// TIA Portal V17 export
// export: Created 2021-12-03T08:13:11.653875Z, ExportSetting WithDefaults, DisplayName Totally Integrated Automation Portal, DisplayVersion V17, DisplayName TIA Portal Openness, DisplayVersion V17, DisplayName TIA Portal Version Control Interface, DisplayVersion V17, DisplayName STEP 7 Professional, DisplayVersion V17, DisplayName STEP 7 Safety, DisplayVersion V17, DisplayName WinCC Advanced, DisplayVersion V17
FUNCTION "FFC_ContCtrl" : Void   // FC700, F_FBD
VERSION : 0.1
// stored: AutoNumber false, IsIECCheckEnabled false, UDAEnableTagReadback false
BEGIN

REGION Network 2: Таймер на включение 400В через 15 секунд после 230В / Задержка между включением 230 и 380 В
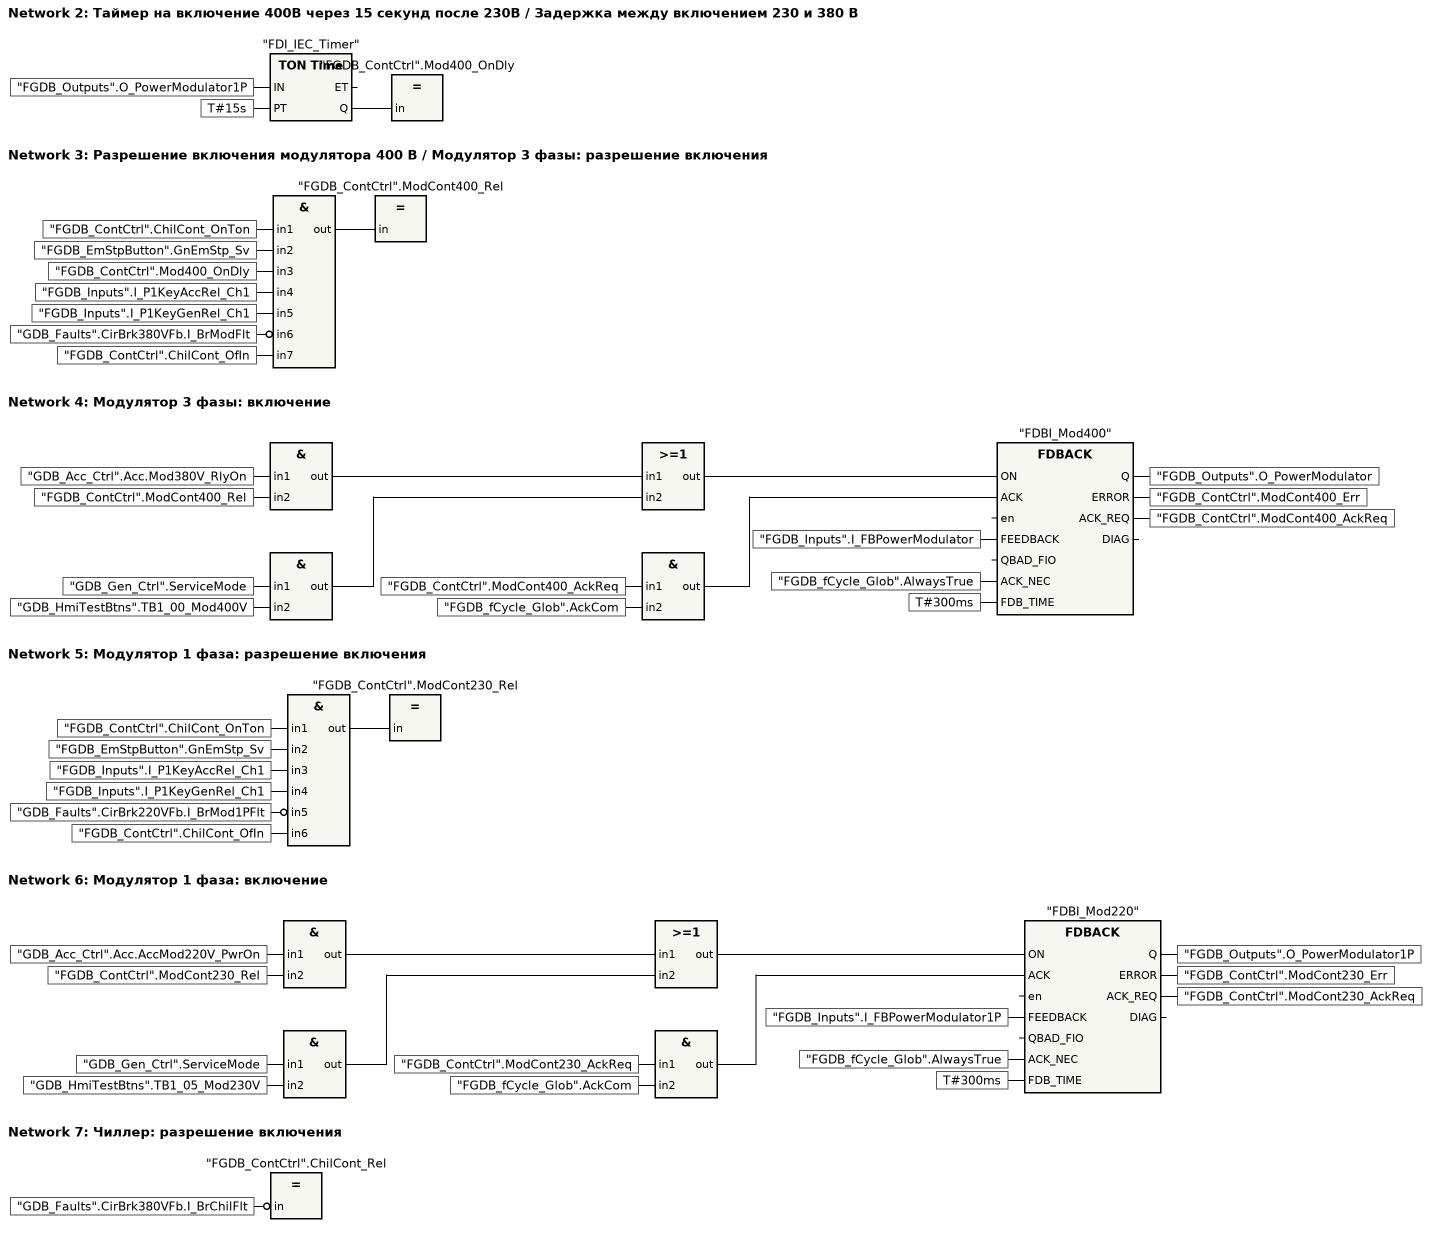
   "FDI_IEC_Timer".TON(IN := "FGDB_Outputs".O_PowerModulator1P, PT := T#15s);
   "FGDB_ContCtrl".Mod400_OnDly := "FDI_IEC_Timer".Q;
END_REGION

REGION Network 3: Разрешение включения модулятора 400 В / Модулятор 3 фазы: разрешение включения
   "FGDB_ContCtrl".ModCont400_Rel := "FGDB_ContCtrl".ChilCont_OnTon AND "FGDB_EmStpButton".GnEmStp_Sv AND "FGDB_ContCtrl".Mod400_OnDly AND "FGDB_Inputs".I_P1KeyAccRel_Ch1 AND "FGDB_Inputs".I_P1KeyGenRel_Ch1 AND NOT "GDB_Faults".CirBrk380VFb.I_BrModFlt AND "FGDB_ContCtrl".ChilCont_OfIn;
END_REGION

REGION Network 4: Модулятор 3 фазы: включение
   "FDBI_Mod400"(ON := ("GDB_Acc_Ctrl".Acc.Mod380V_RlyOn AND "FGDB_ContCtrl".ModCont400_Rel) OR ("GDB_Gen_Ctrl".ServiceMode AND "GDB_HmiTestBtns".TB1_00_Mod400V),   // FDBACK
                 ACK := "FGDB_ContCtrl".ModCont400_AckReq AND "FGDB_fCycle_Glob".AckCom,
                 FEEDBACK := "FGDB_Inputs".I_FBPowerModulator,
                 ACK_NEC := "FGDB_fCycle_Glob".AlwaysTrue,
                 FDB_TIME := T#300ms,
                 Q => "FGDB_Outputs".O_PowerModulator,
                 ERROR => "FGDB_ContCtrl".ModCont400_Err,
                 ACK_REQ => "FGDB_ContCtrl".ModCont400_AckReq);
END_REGION

REGION Network 5: Модулятор 1 фаза: разрешение включения
   "FGDB_ContCtrl".ModCont230_Rel := "FGDB_ContCtrl".ChilCont_OnTon AND "FGDB_EmStpButton".GnEmStp_Sv AND "FGDB_Inputs".I_P1KeyAccRel_Ch1 AND "FGDB_Inputs".I_P1KeyGenRel_Ch1 AND NOT "GDB_Faults".CirBrk220VFb.I_BrMod1PFlt AND "FGDB_ContCtrl".ChilCont_OfIn;
END_REGION

REGION Network 6: Модулятор 1 фаза: включение
   "FDBI_Mod220"(ON := ("GDB_Acc_Ctrl".Acc.AccMod220V_PwrOn AND "FGDB_ContCtrl".ModCont230_Rel) OR ("GDB_Gen_Ctrl".ServiceMode AND "GDB_HmiTestBtns".TB1_05_Mod230V),   // FDBACK
                 ACK := "FGDB_ContCtrl".ModCont230_AckReq AND "FGDB_fCycle_Glob".AckCom,
                 FEEDBACK := "FGDB_Inputs".I_FBPowerModulator1P,
                 ACK_NEC := "FGDB_fCycle_Glob".AlwaysTrue,
                 FDB_TIME := T#300ms,
                 Q => "FGDB_Outputs".O_PowerModulator1P,
                 ERROR => "FGDB_ContCtrl".ModCont230_Err,
                 ACK_REQ => "FGDB_ContCtrl".ModCont230_AckReq);
END_REGION

REGION Network 7: Чиллер: разрешение включения
   "FGDB_ContCtrl".ChilCont_Rel := NOT "GDB_Faults".CirBrk380VFb.I_BrChilFlt;
END_REGION

REGION Network 8: Чиллер: выбор времени выключения
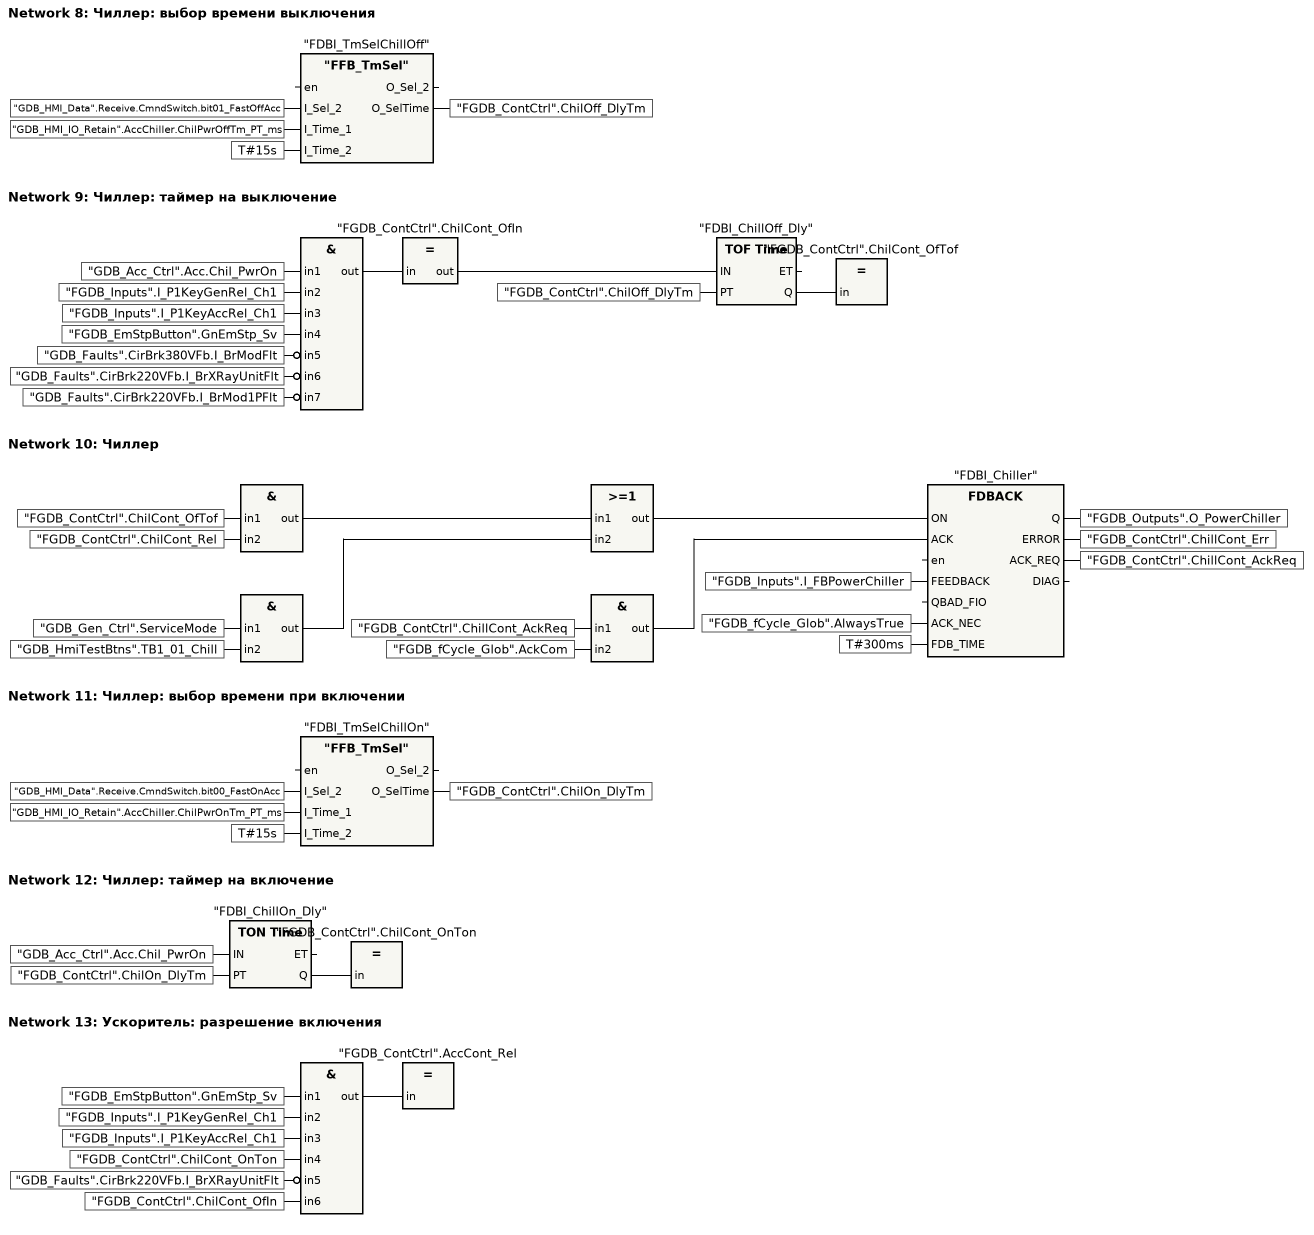
   "FDBI_TmSelChillOff"(I_Sel_2 := "GDB_HMI_Data".Receive.CmndSwitch.bit01_FastOffAcc,   // "FFB_TmSel"
                        I_Time_1 := "GDB_HMI_IO_Retain".AccChiller.ChilPwrOffTm_PT_ms,
                        I_Time_2 := T#15s,
                        O_SelTime => "FGDB_ContCtrl".ChilOff_DlyTm);
END_REGION

REGION Network 9: Чиллер: таймер на выключение
   "FGDB_ContCtrl".ChilCont_OfIn := "GDB_Acc_Ctrl".Acc.Chil_PwrOn AND "FGDB_Inputs".I_P1KeyGenRel_Ch1 AND "FGDB_Inputs".I_P1KeyAccRel_Ch1 AND "FGDB_EmStpButton".GnEmStp_Sv AND NOT "GDB_Faults".CirBrk380VFb.I_BrModFlt AND NOT "GDB_Faults".CirBrk220VFb.I_BrXRayUnitFlt AND NOT "GDB_Faults".CirBrk220VFb.I_BrMod1PFlt;
   "FDBI_ChillOff_Dly".TOF(IN := "FGDB_ContCtrl".ChilCont_OfIn, PT := "FGDB_ContCtrl".ChilOff_DlyTm);
   "FGDB_ContCtrl".ChilCont_OfTof := "FDBI_ChillOff_Dly".Q;
END_REGION

REGION Network 10: Чиллер
   "FDBI_Chiller"(ON := ("FGDB_ContCtrl".ChilCont_OfTof AND "FGDB_ContCtrl".ChilCont_Rel) OR ("GDB_Gen_Ctrl".ServiceMode AND "GDB_HmiTestBtns".TB1_01_Chill),   // FDBACK
                  ACK := "FGDB_ContCtrl".ChillCont_AckReq AND "FGDB_fCycle_Glob".AckCom,
                  FEEDBACK := "FGDB_Inputs".I_FBPowerChiller,
                  ACK_NEC := "FGDB_fCycle_Glob".AlwaysTrue,
                  FDB_TIME := T#300ms,
                  Q => "FGDB_Outputs".O_PowerChiller,
                  ERROR => "FGDB_ContCtrl".ChillCont_Err,
                  ACK_REQ => "FGDB_ContCtrl".ChillCont_AckReq);
END_REGION

REGION Network 11: Чиллер: выбор времени при включении
   "FDBI_TmSelChillOn"(I_Sel_2 := "GDB_HMI_Data".Receive.CmndSwitch.bit00_FastOnAcc,   // "FFB_TmSel"
                       I_Time_1 := "GDB_HMI_IO_Retain".AccChiller.ChilPwrOnTm_PT_ms,
                       I_Time_2 := T#15s,
                       O_SelTime => "FGDB_ContCtrl".ChilOn_DlyTm);
END_REGION

REGION Network 12: Чиллер: таймер на включение
   "FDBI_ChillOn_Dly".TON(IN := "GDB_Acc_Ctrl".Acc.Chil_PwrOn, PT := "FGDB_ContCtrl".ChilOn_DlyTm);
   "FGDB_ContCtrl".ChilCont_OnTon := "FDBI_ChillOn_Dly".Q;
END_REGION

REGION Network 13: Ускоритель: разрешение включения
   "FGDB_ContCtrl".AccCont_Rel := "FGDB_EmStpButton".GnEmStp_Sv AND "FGDB_Inputs".I_P1KeyGenRel_Ch1 AND "FGDB_Inputs".I_P1KeyAccRel_Ch1 AND "FGDB_ContCtrl".ChilCont_OnTon AND NOT "GDB_Faults".CirBrk220VFb.I_BrXRayUnitFlt AND "FGDB_ContCtrl".ChilCont_OfIn;
END_REGION

REGION Network 14: Ускоритель: включение
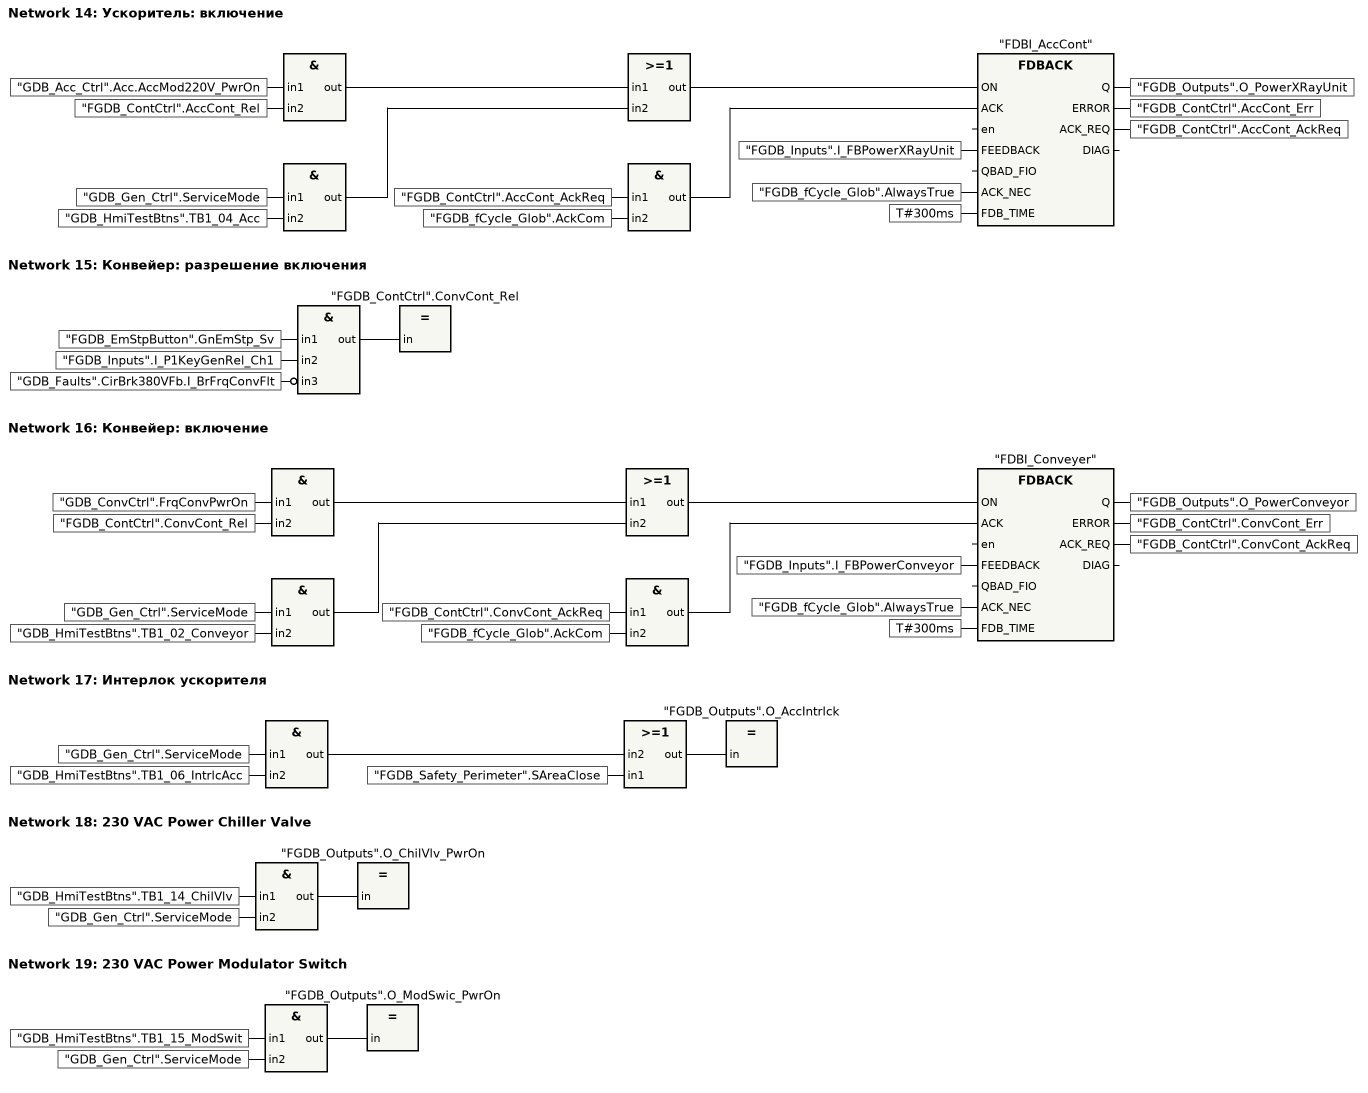
   "FDBI_AccCont"(ON := ("GDB_Acc_Ctrl".Acc.AccMod220V_PwrOn AND "FGDB_ContCtrl".AccCont_Rel) OR ("GDB_Gen_Ctrl".ServiceMode AND "GDB_HmiTestBtns".TB1_04_Acc),   // FDBACK
                  ACK := "FGDB_ContCtrl".AccCont_AckReq AND "FGDB_fCycle_Glob".AckCom,
                  FEEDBACK := "FGDB_Inputs".I_FBPowerXRayUnit,
                  ACK_NEC := "FGDB_fCycle_Glob".AlwaysTrue,
                  FDB_TIME := T#300ms,
                  Q => "FGDB_Outputs".O_PowerXRayUnit,
                  ERROR => "FGDB_ContCtrl".AccCont_Err,
                  ACK_REQ => "FGDB_ContCtrl".AccCont_AckReq);
END_REGION

REGION Network 15: Конвейер: разрешение включения
   "FGDB_ContCtrl".ConvCont_Rel := "FGDB_EmStpButton".GnEmStp_Sv AND "FGDB_Inputs".I_P1KeyGenRel_Ch1 AND NOT "GDB_Faults".CirBrk380VFb.I_BrFrqConvFlt;
END_REGION

REGION Network 16: Конвейер: включение
   "FDBI_Conveyer"(ON := ("GDB_ConvCtrl".FrqConvPwrOn AND "FGDB_ContCtrl".ConvCont_Rel) OR ("GDB_Gen_Ctrl".ServiceMode AND "GDB_HmiTestBtns".TB1_02_Conveyor),   // FDBACK
                   ACK := "FGDB_ContCtrl".ConvCont_AckReq AND "FGDB_fCycle_Glob".AckCom,
                   FEEDBACK := "FGDB_Inputs".I_FBPowerConveyor,
                   ACK_NEC := "FGDB_fCycle_Glob".AlwaysTrue,
                   FDB_TIME := T#300ms,
                   Q => "FGDB_Outputs".O_PowerConveyor,
                   ERROR => "FGDB_ContCtrl".ConvCont_Err,
                   ACK_REQ => "FGDB_ContCtrl".ConvCont_AckReq);
END_REGION

REGION Network 17: Интерлок ускорителя
   "FGDB_Outputs".O_AccIntrlck := ("GDB_Gen_Ctrl".ServiceMode AND "GDB_HmiTestBtns".TB1_06_IntrlcAcc) OR "FGDB_Safety_Perimeter".SAreaClose;
END_REGION

REGION Network 18: 230 VAC Power Chiller Valve
   "FGDB_Outputs".O_ChilVlv_PwrOn := "GDB_HmiTestBtns".TB1_14_ChilVlv AND "GDB_Gen_Ctrl".ServiceMode;
END_REGION

REGION Network 19: 230 VAC Power Modulator Switch
   "FGDB_Outputs".O_ModSwic_PwrOn := "GDB_HmiTestBtns".TB1_15_ModSwit AND "GDB_Gen_Ctrl".ServiceMode;
END_REGION
END_FUNCTION
